// Block: A0302_HU_Cytropack_PERS

DATA_BLOCK A0302_HU_Cytropack_PERS
VERSION : 0.1
   NON_RETAIN
   VAR
      Par : Struct
         Bloccaggio : Struct
            TargetPressure : Real;
            TargetMaxSpeed : Real;
            Delta : Struct
               Min : Real;
               Max : Real;
            END_STRUCT;
         END_STRUCT;
         Pareggiamento : Struct
            TargetPressure : Real;
            TargetMaxSpeed : Real;
            Delta : Struct
               Min : Real;
               Max : Real;
            END_STRUCT;
         END_STRUCT;
      END_STRUCT;
   END_VAR

BEGIN
   // No initialization required
END_DATA_BLOCK
